// TIA Portal V20 export
FUNCTION_BLOCK "LER_CM_Name"   // FB89, LAD
// stored: Access Published, MemoryReserve 100, SetENOAutomatically false
   VAR_INPUT
      Read : Bool;
      Write : Bool;
      StartArr : Int;
      CntAr : Int;
   END_VAR
   VAR_IN_OUT
      HMIAxis_1 : WString;
      HMIAxis_2 : WString;
      HMIAxis_3 : WString;
      HMIAxis_4 : WString;
      HMIAxis_5 : WString;
      Config_1 : WString;
      Config_2 : WString;
      Config_3 : WString;
      Config_4 : WString;
      Config_5 : WString;
      NameManDB : Array[*] of WString [25];
   END_VAR
   VAR
      Temp : WString[25];
      AxisBuffer : Array[1..5] of WString[25];
      EndCnt : Int;
      i : Int;
      S : Int;
      P : Array[0..7] of Bool;
   END_VAR
BEGIN

REGION Network 2 (SCL)
   #P[0] :=#Read AND NOT #P[1] ;
   #P[1] :=#Read;

   #P[2] :=#Write AND NOT #P[3] ;
   #P[3] := #Write;

   #S := #StartArr;

   IF #S > 0 THEN

       IF #CntAr <= 5 THEN
           #EndCnt := #CntAr;

       ELSE
           #EndCnt := 5;
       END_IF;

       IF #P[0] THEN
           #AxisBuffer[1] := #HMIAxis_1;
           #AxisBuffer[2] := #HMIAxis_2;
           #AxisBuffer[3] := #HMIAxis_3;
           #AxisBuffer[4] := #HMIAxis_4;
           #AxisBuffer[5] := #HMIAxis_5;

           FOR #i := 1 TO #EndCnt DO
               ;

               #NameManDB[#S] := #AxisBuffer[#i];
               #S := #S + 1;

           END_FOR;
       END_IF;

       IF #P[2] THEN

           FOR #i := 1 TO #EndCnt DO
               ;
               #AxisBuffer[#i] := #NameManDB[#S];
               #S := #S + 1;

           END_FOR;

           #HMIAxis_1 := #Config_1 := #AxisBuffer[1];
           #HMIAxis_2 := #Config_2 := #AxisBuffer[2];
           #HMIAxis_3 := #Config_3 := #AxisBuffer[3];
           #HMIAxis_4 := #Config_4 := #AxisBuffer[4];
           #HMIAxis_5 := #Config_5 := #AxisBuffer[5];
       END_IF;
   END_IF;
END_REGION
END_FUNCTION_BLOCK
